			IF nEcSlaveState.3					(* Slave in OP *)
				AND tCoEReadCycle <> T#0MS 		(* tCoEReadCycle <> t#0ms -> Read diagnostic aktiv *)
			THEN
				bReadDiagObjError := FALSE;
				fbEcCoeSdoRead(	bExecute := FALSE);
				fbTimer(IN := FALSE);
				eReadDiagObjState := eCycleDiagObj_ReadTemperature;
			END_IF

			
		eCycleDiagObj_ReadTemperature	:	(* Read temperature *)

			fbEcCoeSdoRead(
				sNetId			:= 	F_CreateAmsNetId(stEcAdsAddr.netId),
				nSlaveAddr		:= 	stEcAdsAddr.port,
				nSubIndex		:= 	1,
				nIndex			:= 	16#F984,
				pDstBuf			:= 	ADR(stTsSlaveInfo.stTsDiagObjectsBitsEL2912[1]),
				cbBufLen		:= 	SIZEOF(stTsSlaveInfo.stTsDiagObjectsBitsEL2912[1]),
				bExecute		:= 	TRUE,
				tTimeout		:= 	DEFAULT_ADS_TIMEOUT,
				bCompleteAccess	:= 	TRUE);

			IF NOT fbEcCoeSdoRead.bBusy 
				AND NOT fbEcCoeSdoRead.bError 
			THEN
				fbEcCoeSdoRead(bExecute := FALSE);
				eReadDiagObjState := eCycleDiagObj_ReadDiag;
			ELSIF NOT fbEcCoeSdoRead.bBusy 
				AND fbEcCoeSdoRead.bError 
			THEN
				eReadDiagObjErrStep := eReadDiagObjState;
				eReadDiagObjState 	:= eCycleDiagObj_Error;
			END_IF

			
		eCycleDiagObj_ReadDiag			:	(* Read diacnostic objects *)

			fbTimer(IN := TRUE, PT := tCoEReadCycle);
			fbEcCoeSdoRead(
				sNetId			:= 	F_CreateAmsNetId(stEcAdsAddr.netId),
				nSlaveAddr		:= 	stEcAdsAddr.port,
				nSubIndex		:= 	1,
				nIndex			:= 	16#F985,
				pDstBuf			:= 	ADR(stTsSlaveInfo.stTsDiagObjectsBitsEL2912[2]),
				cbBufLen		:= 	SIZEOF(stTsSlaveInfo.stTsDiagObjectsBitsEL2912[2]),
				bExecute		:= 	TRUE,
				tTimeout		:= 	DEFAULT_ADS_TIMEOUT,
				bCompleteAccess	:= 	TRUE);

			IF NOT fbEcCoeSdoRead.bBusy 
				AND NOT fbEcCoeSdoRead.bError 
			THEN
				fbEcCoeSdoRead(bExecute := FALSE);
				eReadDiagObjState := eCycleDiagObj_ReadDelay;
			ELSIF NOT fbEcCoeSdoRead.bBusy 
				AND fbEcCoeSdoRead.bError 
			THEN
				eReadDiagObjErrStep := eReadDiagObjState;
				eReadDiagObjState 	:= eCycleDiagObj_Error;
			END_IF
			
			
		eCycleDiagObj_ReadDelay		:	(* Read delay *)
			fbTimer(
				IN := TRUE, 
				PT := tCoEReadCycle);

			IF fbTimer.Q 
			THEN
				fbTimer(IN := FALSE); 			
				eReadDiagObjState := eCycleDiagObj_Done;
			END_IF

			
		eCycleDiagObj_Done				:	(* Done *)

			eReadDiagObjState := eCycleDiagObj_Init;

			
		eCycleDiagObj_Error			:	(* Error detected *)

			bReadDiagObjError := TRUE;
		
			IF bReadDiagObjReset
			THEN
				bReadDiagObjError := FALSE;
				fbEcCoeSdoRead(bExecute := FALSE);
				eReadDiagObjErrStep := E_TsCycleDiagObj.eCycleDiagObj_NoError;
				eReadDiagObjState := eCycleDiagObj_Init;
			END_IF

	ELSE
		
		eReadDiagObjState := eCycleDiagObj_Init;
		
	END_CASE
	stTsSlaveInfo.stSlaveTemp.nInternalTemperature1 := stTsSlaveInfo.stTsDiagObjectsBitsEL2912[1].nTemperatureC;
	stTsSlaveInfo.stSlaveTemp.nInternalTemperature2 := stTsSlaveInfo.stTsDiagObjectsBitsEL2912[2].nTemperatureC;	

	stTsSlaveInfo.bIntTempWarning1 := stTsSlaveInfo.stSlaveTemp.nInternalTemperature1 >= nWarningLevelTemp1;
	stTsSlaveInfo.bIntTempWarning2 := stTsSlaveInfo.stSlaveTemp.nInternalTemperature2 >= nWarningLevelTemp2;

(* End *)
END_ACTION

ACTION act_Signals:
(* Evaluate the EL2912 signals *)

	IF nEcSlaveState.3 (* Slave in operational state *)
	THEN

		(* OP -> transfer the signal states *)
		
		stTsSlaveInfo.bFSOUTModule1Fault 	:= stInfoData.nInOutSafeDataByte1.0;
		stTsSlaveInfo.bFSOUTModule2Fault  	:= stInfoData.nInOutSafeDataByte1.1;	
		
		stTsSlaveInfo.bFSOUTChannel1 		:= stInfoData.nInOutSafeDataByte2.0;	
		stTsSlaveInfo.bFSOUTChannel2 	  	:= stInfoData.nInOutSafeDataByte2.2;
		stTsSlaveInfo.bFSOUTModule1ErrAck  	:= stInfoData.nInOutSafeDataByte2.1;			
		stTsSlaveInfo.bFSOUTModule2ErrAck 	:= stInfoData.nInOutSafeDataByte2.3;
	
ELSE

		(* Error -> clear the signal states *)
		stTsSlaveInfo.bFSOUTModule1Fault  	:= FALSE;
		stTsSlaveInfo.bFSOUTModule2Fault  	:= FALSE;
		stTsSlaveInfo.bFSOUTChannel1  		:= FALSE; 
		stTsSlaveInfo.bFSOUTChannel2  		:= FALSE;
		stTsSlaveInfo.bFSOUTChannel1 		:= FALSE;
		
		stTsSlaveInfo.bFSOUTModule1ErrAck  	:= FALSE;
		stTsSlaveInfo.bFSOUTModule2ErrAck 	:= FALSE;

		
	END_IF

(* End *)
END_ACTION

END_FUNCTION_BLOCK

// ---- POUs/TwinSAFE/FB_EcGetSlaveName.TcPOU
FUNCTION_BLOCK FB_EcGetSlaveName
(*******************************************************************************************************
Title				:	Get EtherCAT slave name
Description			:	Read the EtherCAT slave name from the EtherCAT Master CoE table
Version / Date		:	1.0.0 / 23.05.2016 / created program (Version progress see below)
********************************************************************************************************)
VAR_INPUT

	bExecute                        		:BOOL;							(* The block is activated by a rising edge at this input *)
	sNetId          						:T_AmsNetId;					(* AmsNetId of the EtherCAT master device *)
	nSlaveAddr      						:UINT; 							(* Address of the slave device *)
	tTimeout                        		:TIME := DEFAULT_ADS_TIMEOUT;

END_VAR
VAR_OUTPUT

	bBusy           						:BOOL;							(* This output is set when the function block is activated *)
	sSlaveName         						:STRING[31];					(* Name of this EtherCAT Slave *)
	bError          						:BOOL;
	nErrId          						:UDINT;

END_VAR
VAR

	eStateEcGetSlaveNameSeq					:E_EcGetSlaveName;
	eEcGetSlaveNameErrStep					:E_EcGetSlaveName := eEcGetSlaveName_NoError;

	fbEcGetAllSlaveAddr						:FB_EcGetAllSlaveAddr;
	aAllSlaveAddr							:ARRAY[cMinNumberEcSlaves..cMaxNumberEcSlaves] OF UINT;
	nSlaveAddrIndex							:UINT;
	fbEcCoeSdoRead							:FB_EcCoESdoReadEx;

END_VAR
VAR CONSTANT

	cMinNumberEcSlaves						:UINT := 0;
	cMaxNumberEcSlaves						:UINT := 100;

END_VAR
(*******************************************************************************************************
Version / Date / Description:
1.0.0   / 23.05.2016 / created program
********************************************************************************************************)
(* End *)

(* FB_EcGetSlaveName *)

	CASE eStateEcGetSlaveNameSeq OF 
	
		eEcGetSlaveName_Start				:	(* Waiting for start *)
			
			IF bExecute
			THEN
				bBusy := TRUE;
				eStateEcGetSlaveNameSeq := eEcGetSlaveName_Init;
			END_IF
		
		eEcGetSlaveName_Init				:	(* Initialize functions *)

			fbEcGetAllSlaveAddr(bExecute := FALSE);
			fbEcCoeSdoRead(		bExecute := FALSE);
			
			eStateEcGetSlaveNameSeq := eEcGetSlaveName_ReadAllSlaveAddr;
			
	
		eEcGetSlaveName_ReadAllSlaveAddr	:	(* Read all EtherCAT Slave addresses and find the slave position in the EtherCAT bus *)

			fbEcGetAllSlaveAddr(
				sNetId	 := sNetId, 
				pAddrBuf := ADR(aAllSlaveAddr), 
				cbBufLen := SIZEOF(aAllSlaveAddr), 
				bExecute := TRUE, 
				tTimeout := DEFAULT_ADS_TIMEOUT);

			IF NOT fbEcGetAllSlaveAddr.bBusy
				AND NOT fbEcGetAllSlaveAddr.bError
			THEN
			
				FOR nSlaveAddrIndex := cMinNumberEcSlaves TO cMaxNumberEcSlaves BY 1 DO
					IF nSlaveAddr = aAllSlaveAddr[nSlaveAddrIndex]
					THEN
						EXIT;
					END_IF
				END_FOR

				fbEcGetAllSlaveAddr(bExecute := FALSE);
			
				eStateEcGetSlaveNameSeq := eEcGetSlaveName_ReadSlaveName;
	
			ELSIF NOT fbEcGetAllSlaveAddr.bBusy
				AND fbEcGetAllSlaveAddr.bError
			THEN

				nErrId					:=	fbEcGetAllSlaveAddr.nErrId;
				eEcGetSlaveNameErrStep	:= 	eStateEcGetSlaveNameSeq;
				eStateEcGetSlaveNameSeq := 	eEcGetSlaveName_ErrorStep;
			
			END_IF

		eEcGetSlaveName_ReadSlaveName		:	(* Read the EtherCAT slave name from the EtherCAT master CoE table *)
				
			fbEcCoeSdoRead(
				sNetId		:= sNetId, 
				nSlaveAddr	:= 16#FFFF, 						(* EtherCAT master address = 16#FFFF *)
				nSubIndex	:= 3, 
				nIndex		:= 16#8000 + nSlaveAddrIndex, 
				pDstBuf		:= ADR(sSlaveName), 
				cbBufLen	:= SIZEOF(sSlaveName), 
				bExecute	:= TRUE, 
				tTimeout	:= DEFAULT_ADS_TIMEOUT);	


			IF NOT fbEcCoeSdoRead.bBusy
				AND NOT fbEcCoeSdoRead.bError
			THEN
					
				fbEcCoeSdoRead(bExecute := FALSE);

				eStateEcGetSlaveNameSeq := eEcGetSlaveName_Done;
	
			ELSIF NOT fbEcCoeSdoRead.bBusy
				AND fbEcCoeSdoRead.bError
			THEN
				nErrId					:=	fbEcCoeSdoRead.nErrId;
				eEcGetSlaveNameErrStep	:= 	eStateEcGetSlaveNameSeq;
				eStateEcGetSlaveNameSeq := 	eEcGetSlaveName_ErrorStep;
			
			END_IF


		eEcGetSlaveName_Done				:	(* EtherCAT slave name read done *)

			bBusy := FALSE;

			IF NOT bExecute
			THEN
				eStateEcGetSlaveNameSeq := eEcGetSlaveName_Start;
			END_IF

		eEcGetSlaveName_ErrorStep			:	(* Error detected *)

			bBusy := FALSE;
			bError := TRUE;

			IF NOT bExecute
			THEN
				fbEcGetAllSlaveAddr(bExecute 	:= FALSE);
				fbEcCoeSdoRead(		bExecute 	:= FALSE);
				
				bError 							:= FALSE;
				nErrId 							:= 0;
				
				eStateEcGetSlaveNameSeq 		:= eEcGetSlaveName_Start;
				eEcGetSlaveNameErrStep			:= eEcGetSlaveName_NoError;
			END_IF
		
	ELSE

		eStateEcGetSlaveNameSeq := eEcGetSlaveName_Start;
		eEcGetSlaveNameErrStep	:= eEcGetSlaveName_NoError;
	
	END_CASE

(* End *)

END_FUNCTION_BLOCK

// ---- POUs/VISION.TcPOU
PROGRAM VISION
VAR
	hr					: HRESULT;
	bActivateVisionAcqu AT %I*: BOOL;
	bDeactivateVisionAcqu AT %I*: BOOL;
	bActiveState : BOOL;
	fbControl			: FB_VN_SimpleCameraControl;
	eState				: ETcVnCameraState;
	
	// Image
	ipImage				: ITcVnImage;
	ipImageWork			: ITcVnImage;
	ipImageResult		: ITcVnImage;
	
	// displayable Image
	ipImageDispl		: ITcVnDisplayableImage;
	ipImageWorkDispl	: ITcVnDisplayableImage;
	ipImageResultDispl	: ITcVnDisplayableImage;
//											[R , G , B , L]
	aLowerBounds		: TcVnVector4_LREAL :=[30,45,90,0];
	aUpperBounds		: TcVnVector4_LREAL :=[50,80,255,0];
	
	ipContours			: ITcVnContainer;
	nNumberofElements	: ULINT;
	
	aColorRed			: TcVnVector4_LREAL :=[255,0,0,0];
	aColorGreen			: TcVnVector4_LREAL :=[0,255,0,0];
	
	ipIterator			: ITcVnForwardIterator;
	ipContoursSingle	: ITcVnContainer;
	fArea				: LREAL;
	
	aCenterOfMass		: TcVnPoint2_LREAL;
	stRectangle			: TcVnRotatedRectangle;
END_VAR

// Detect activate/deactivate state for function 
IF 	bActivateVisionAcqu AND NOT bDeactivateVisionAcqu THEN
	bActiveState:=TRUE;
ELSIF
	bDeactivateVisionAcqu AND NOT bActivateVisionAcqu THEN
	bActiveState:=FALSE;
END_IF

eState := fbControl.GetState();

CASE eState OF
	TCVN_CS_INITIAL, 			(* The camera controller is in the initial state and ready to establish the connection to the camera. *)
	TCVN_CS_INITIALIZING, 		(* The camera controller is initializing the camera. *)
	TCVN_CS_INITIALIZED, 		(* The camera controller has initialized the camera. *)
	TCVN_CS_OPENING, 			(* The camera controller is establishing the connection to the camera. *)
	TCVN_CS_OPENED, 			(* The connection to the camera has been established and the camera controller is ready to start the image acquisition. *)
	TCVN_CS_STARTACQUISITION: 	(* The camera controller is starting the image acquisition. *)
	
		hr := fbControl.StartAcquisition();
	
	TCVN_CS_ACQUIRING: 			(* The camera is sending images (either streaming or manually triggered, depending on the configuration). *)
		IF bActiveState THEN
			hr := fbControl.GetCurrentImage(ipImage);
		END_IF
		IF SUCCEEDED(hr) THEN
			
			// debug *
			hr := F_VN_CopyIntoDisplayableImage(ipSrcImage:= ipImage, ipDestImage:= ipImageDispl, hrPrev:= hr) ; 
			
			// convert color space
			hr := F_VN_ConvertColorSpace(ipSrcImage:= ipImage, 
										ipDestImage:= ipImageWork, 
										eTransform:= ETcVnColorSpaceTransform.TCVN_CST_BAYER_RG_TO_RGB, 
										hrPrev:= hr);
										
			//// copyImage
			hr := F_VN_CopyImage(ipImageWork,ipImageResult,hr);
										
			// Debug **
			//hr := F_VN_CopyIntoDisplayableImage(ipSrcImage:= ipImageWork, ipDestImage:= ipImageWorkDispl, hrPrev:= hr) ;
			
			// CheckColorRange
			hr := F_VN_CheckColorRange(
										ipSrcImage:= ipImageWork, 
										ipDestImage:= ipImageWork, 
										aLowerBounds:= aLowerBounds, 
										aUpperBounds:= aUpperBounds, 
										hrPrev:= hr);
			
			// Debug **
			hr := F_VN_CopyIntoDisplayableImage(ipSrcImage:= ipImageWork, ipDestImage:= ipImageWorkDispl, hrPrev:= hr) ;
			
			// FindContours
			hr := F_VN_FindContours(ipSrcImage:= ipImageWork, ipContours:= ipContours, hrPrev:= hr);
			
			//nNumberofElements := ipContours.GetElementNum(); wrong way
			hr := F_VN_GetNumberOfElements(ipContainer:= ipContours, nNumberOfElements:= nNumberofElements, hrPrev:= hr);
	
//////-----------------------------
			// LOOP
			hr := F_VN_GetForwardIterator(ipContainer:= ipContours, ipIterator:= ipIterator, hrPrev:= hr);
			
			WHILE SUCCEEDED(hr) AND_THEN ipIterator.CheckIfEnd() <> S_OK DO
				
				// getContainer
				hr := F_VN_GetContainer(ipIterator:= ipIterator, ipContainer:= ipContoursSingle, hrPrev:= hr);
				hr := F_VN_IncrementIterator(ipIterator,hr); // !!!!!!
				
				//------------------------------------------
				
				hr := F_VN_ContourArea(ipContoursSingle,fArea,hr);
				
				IF fArea > 50_000 AND fArea < 400_000 THEN
					
					//// DrawContours
					hr := F_VN_DrawContours(
										ipContours:= ipContoursSingle, // !!!
										nContourIndex:= -1, 
										ipDestImage:= ipImageResult, 
										aColor:= aColorRed, 
										nThickness:= 5, 
										hrPrev:= hr);
										
//					F_VN_ContourCenterOfMass
					hr := F_VN_ContourCenterOfMass(ipContour:= ipContoursSingle, 
													aCenterOfMass:= aCenterOfMass, 
													hrPrev:= hr);
//					F_VN_DrawPointExp
					hr := F_VN_DrawPointExp(
											nX:= TO_UDINT(aCenterOfMass[0]), 
											nY:= TO_UDINT(aCenterOfMass[1]), 
											ipDestImage:= ipImageResult, 
											eShape:= ETcVnDrawShape.TCVN_DS_X, 
											aColor:= aColorGreen, 
											nSize:= 20, //5
											nThickness:= 5, 
											eLineType:= ETcVnLineType.TCVN_LT_4_CONNECTED, 
											hrPrev:= hr);
//					F_VN_EnclosingRectangle
					hr := F_VN_EnclosingRectangle(ipPointSet:= ipContoursSingle, stRectangle:= stRectangle, hrPrev:= hr);
//					F_VN_DrawRotatedRectangle
					hr := F_VN_DrawRotatedRectangle(
											stRectangle:= stRectangle, 
											ipDestImage:= ipImageResult, 
											aColor:= aColorRed, 
											nThickness:= 5, 
											hrPrev:= hr);
//					F_VN_PutTextExp
					hr := F_VN_PutTextExp(
											sText:= 'BLUE', 
											ipDestImage:= ipImageResult, 
											nX:= TO_UDINT(stRectangle.aCenter[0] - stRectangle.stSize.fHeight/2), 
											nY:= TO_UDINT(stRectangle.aCenter[1] - stRectangle.stSize.fHeight/2), 
											eFontType:= ETcVnFontType.TCVN_FT_HERSHEY_COMPLEX, 
											fFontScale:= 5, 
											aColor:= aColorRed, 
											nThickness:= 5, 
											eLineType:= ETcVnLineType.TCVN_LT_4_CONNECTED, 
											bBottomLeftOrigin:= FALSE, 
											hrPrev:= hr);
					
				END_IF
				
			END_WHILE

//////-----------------------------

			//// DrawContours
//			hr := F_VN_DrawContours(
//									ipContours:= ipContours, 
//									nContourIndex:= -1, 
//									ipDestImage:= ipImageResult, 
//									aColor:= aColorRed, 
//									nThickness:= 5, 
//									hrPrev:= hr);
			
			// Debug ** copy need time & memory & just 1 side can access the image | transform: save time
			//hr := F_VN_CopyIntoDisplayableImage(ipSrcImage:= ipImageResult, ipDestImage:= ipImageResultDispl, hrPrev:= hr);
			hr := F_VN_TransformIntoDisplayableImageExp(ipSrcImage:= ipImageResult, ipDestImage:= ipImageResultDispl, bAllowDeepCopy:= TRUE, hrPrev:= hr);
									
		END_IF
		

	TCVN_CS_ERROR: 	(* The camera controller is in an error state (e.g. the connection to the camera was lost). *)
		fbControl.Reset();
END_CASE

END_PROGRAM

// ---- POUs/Vision_test.TcPOU
PROGRAM Vision_test
VAR
	bActivateVisionAcqu AT %I*: BOOL;
	bDeactivateVisionAcqu AT %I*: BOOL;
	bActiveState : BOOL;	

	hr					: HRESULT;
	
	fbControl			: FB_VN_SimpleCameraControl;
	eState				: ETcVnCameraState;
	
	// Image
	ipImage				: ITcVnImage;
	ipImageWork			: ITcVnImage;
	ipImageResult		: ITcVnImage;
	
	// displayable Image
	ipImageDispl		: ITcVnDisplayableImage;
	ipImageWorkDispl	: ITcVnDisplayableImage;
	ipImageResultDispl	: ITcVnDisplayableImage;
	
	// QR Code
	ipCodeDecodedList   :    ITcVnContainer; 
	ipCodeContourList   :    ITcVnContainer;
	sCodeAsString       :    STRING(255);
	sErrorString		:	 STRING(255);
	eBarcodeSearchDirection   :   ETcVnBarcodeSearchDirection := TCVN_BSD_ANY;
	eBarcodeType              :   ETcVnBarcodeType := TCVN_BT_EAN13;


	// Watchdog
	hrWD                :    HRESULT;
	//tStop               :    DINT := 20000; //qr code
	tStop               :    DINT := 50000; //qr code
	tRest               :    DINT;

	// Color
	aRedColor           :    TcVnVector4_LREAL := [255, 0, 0];
	aGreenColor			:	 TcVnVector4_LREAL := [0, 255, 0];

	// Return code
	nReturnCode               :   DWORD;
	sReturnCode               :   STRING;
	sResultText               :   STRING;
END_VAR

// Detect activate/deactivate state for function 
IF 	bActivateVisionAcqu AND NOT bDeactivateVisionAcqu THEN
	bActiveState:=TRUE;
ELSIF
	bDeactivateVisionAcqu AND NOT bActivateVisionAcqu THEN
	bActiveState:=FALSE;
END_IF

eState := fbControl.GetState();

CASE eState OF
	TCVN_CS_INITIAL, 			(* The camera controller is in the initial state and ready to establish the connection to the camera. *)
	TCVN_CS_INITIALIZING, 		(* The camera controller is initializing the camera. *)
	TCVN_CS_INITIALIZED, 		(* The camera controller has initialized the camera. *)
	TCVN_CS_OPENING, 			(* The camera controller is establishing the connection to the camera. *)
	TCVN_CS_OPENED, 			(* The connection to the camera has been established and the camera controller is ready to start the image acquisition. *)
	TCVN_CS_STARTACQUISITION: 	(* The camera controller is starting the image acquisition. *)
	
		hr := fbControl.StartAcquisition();
	
	TCVN_CS_ACQUIRING: 			(* The camera is sending images (either streaming or manually triggered, depending on the configuration). *)
		IF bActiveState THEN
			hr := fbControl.GetCurrentImage(ipImage);
		END_IF
		IF  SUCCEEDED(hr) THEN
			sCodeAsString :='Scanning...';
			// Conver color space from grayscale to RGB, Display input image (without processing)
			hr:=F_VN_ConvertColorSpace(ipImage,ipImageResult,ETcVnColorSpaceTransform.TCVN_CST_GRAY_TO_RGB,hr);
			//hr:= F_VN_CopyImage(ipImage,ipImageResult,hr);
			hr:=F_VN_CopyImage(ipImageResult,ipImageWork,hr);
			hr:= F_VN_CopyIntoDisplayableImage(ipSrcImage:= ipImage,ipDestImage:=ipImageDispl,hrPrev:=hr);
			hr:= F_VN_CopyIntoDisplayableImage(ipSrcImage:= ipImageResult,ipDestImage:=ipImageResultDispl,hrPrev:=hr);
			// Pre result image processing
			hr := F_VN_PutTextExp(sCodeAsString, ipImageWork, 50, 100, TCVN_FT_HERSHEY_PLAIN, 5, aRedColor,3, TCVN_LT_4_CONNECTED, FALSE, hr);
			hr:=F_VN_CopyIntoDisplayableImage(ipSrcImage:= ipImageWork,ipDestImage:=ipImageResultDispl,hrPrev:=hr);

			// Execute the Barcode Reading Function with EAN13 selected monitored by the Watchdog-Function
			hrWD := F_VN_StartRelWatchdog(tStop, hr);
			(*hr := F_VN_ReadQRCodeExp(
            ipSrcImage      :=  ipImage,
            ipDecodedData   :=  ipCodeDecodedList,
            ipContours      :=  ipCodeContourList,
            nCodeNumber     :=  1,
            eSearchStrategy :=  TCVN_CSS_ONLY_NOT_INVERTED + TCVN_CSS_ONLY_NOT_FLIPPED,
            hrPrev          :=  hr
   			 );*)
	    	hr := F_VN_ReadBarcodeExp(
               ipSrcImage         :=   ipImageResult,
               ipDecodedData      :=   ipCodeDecodedList,
               ipContours         :=   ipCodeContourList,
               eBarcodeType       :=   eBarcodeType,
               nCodeNumber        :=   1, 
               eSearchDirection   :=   eBarcodeSearchDirection,
               hrPrev             :=   hr);
			hrWD := F_VN_StopWatchdog(hrWD, tRest => tRest);
			//ADSLOGDINT(msgCtrlMask:=ADSLOG_MSGTYPE_MSGBOX,msgFmtStr:='hrResult1 %d',dintArg:=hr);
			// Handle return-code
			IF hr = S_OK THEN
				// Prepare code result in string
				hr := F_VN_ExportSubContainer_String(ipCodeDecodedList, 0, sCodeAsString, 255, hr);
				sCodeAsString := CONCAT('Code: ', sCodeAsString);
			ELSE
				// Check for succeeded return codes or add specific error handling
				CASE hr OF
					S_FALSE: 
						sCodeAsString := 'No code found...'; 
			
					S_WATCHDOG_TIMEOUT: 
						sCodeAsString := 'Cancelled by watchdog...'; 
				ELSE
					// Extract error-code from HRESULT & react accordingly
					nReturnCode := DINT_TO_DWORD(hr) AND 16#FFF; 
					sReturnCode := DWORD_TO_HEXSTR(nReturnCode, 3, FALSE); 
					sCodeAsString := CONCAT('Returncode ', sReturnCode); 
				END_CASE
			END_IF
			
			// Draw Code Contour into Result Image
		    hr := F_VN_DrawContours(ipCodeContourList, 0, ipImageResult, aGreenColor, 3, hr);
			// Write Code into Result Image
    		hr := F_VN_PutTextExp(sCodeAsString, ipImageResult, 50, 100, TCVN_FT_HERSHEY_PLAIN, 5, aGreenColor,3, TCVN_LT_4_CONNECTED, FALSE, hr);
			// Write Code Reading proceeded time into Result Image
			//sText := CONCAT(CONCAT('Time: ', DINT_TO_STRING(tStop - tRest)), 'us');
			hr := F_VN_TransformIntoDisplayableImage(ipSrcImage:=ipImageResult, ipDestImage:=ipImageResultDispl, hrPrev:=hr);
		END_IF
		

	TCVN_CS_ERROR: 	(* The camera controller is in an error state (e.g. the connection to the camera was lost). *)
		fbControl.Reset();
END_CASE

END_PROGRAM
